// TIA Portal V17 export
// export: Created 2022-04-06T07:28:41.3917177Z, ExportSetting WithDefaults, DisplayName Totally Integrated Automation Portal, DisplayVersion V17, DisplayName TIA Portal Openness, DisplayVersion V17, DisplayName TIA Portal Version Control Interface, DisplayVersion V17, DisplayName TIA Portal Test Suite Advanced, DisplayVersion V17, DisplayName SINAMICS Startdrive Advanced, DisplayVersion V17, DisplayName SINAMICS Startdrive G130, G150, S120, S150, SINAMICS MV, S210, DisplayVersion V17, DisplayName SINAMICS Startdrive G110M, G120, G120C, G120D, G120P, G115D, DisplayVersion V17, DisplayName STEP 7 Professional, DisplayVersion V17, DisplayName STEP 7 Safety, DisplayVersion V17, DisplayName WinCC Advanced / Unified PC, DisplayVersion V17
TYPE "LAxisCtrl_typePhasing"
TITLE = LAxisCtrl_typePhasing
// Support: tech.team.motioncontrol@siemens.com
// stored: IsFailsafeCompliant false
   STRUCT
      phaseShift : LReal := 0.0;   // Absolute or relative leading value shift
      velocity : LReal := -1.0;   // Velocity for leading value shift, added to synchronous operation motion (Value > 0.0: The specified value is used; Value = 0.0: Not permitted; Value < 0.0: Use of the default value configured in the technology object)
      acceleration : LReal := -1.0;   // Acceleration for leading value shift, added to synchronous operation motion (Value > 0.0: The specified value is used; Value = 0.0: Not permitted; Value < 0.0: Use of the default value configured in the technology object)
      deceleration : LReal := -1.0;   // Deceleration for leading value shift, added to synchronous operation motion (Value > 0.0: The specified value is used; Value = 0.0: Not permitted; Value < 0.0: Use of the default value configured in the technology object)
      jerk : LReal := -1.0;   // Jerk for leading value shift, added to synchronous operation motion (Value > 0.0: Smooth velocity profile, the specified value is used; Value = 0.0: Trapezoid velocity profile; Value < 0.0: Use of the default value configured in the technology object)
      phaseAbsolute : Bool := TRUE;   // Indicates the type of phase shift. TRUE: Shift the leading value as an absolute shift; FALSE: Shift the leading value relative to the existing leading value shift
      phaseShiftChangeOnTheFly : Bool := FALSE;   // TRUE: Changing phase shift on-the-fly at absolute phasing; FALSE: Phase shift change requires a new rising edge at phasing input
   END_STRUCT;
END_TYPE
